FUNCTION_BLOCK PAETransport EXTENDS PAModule
VAR_INPUT
END_VAR
VAR_OUTPUT
END_VAR
VAR
	_PAPointMatIn1 : PAPoint(THIS^);
	_PAPointMatOut1 : PAPoint(THIS^);
END_VAR

METHOD FB_init : BOOL
VAR_INPUT
	bInitRetains : BOOL; // if TRUE, the retain variables are initialized (warm start / cold start)
	bInCopyCode : BOOL;  // if TRUE, the instance afterwards gets moved into the copy code (online change)
	parent : IACComponent;
END_VAR
AddPoint(_PAPointMatIn1);
AddPoint(_PAPointMatOut1);
END_METHOD

PROPERTY PUBLIC PAPointMatIn1 : IACPoint
GET
PAPointMatIn1 := _PAPointMatIn1;
END_GET
END_PROPERTY

PROPERTY PUBLIC PAPointMatOut1 : IACPoint
GET
PAPointMatOut1 := _PAPointMatOut1;
END_GET
END_PROPERTY

END_FUNCTION_BLOCK

(* stored: Version 1.1.0.1, ProductVersion 3.1.4020.12
   POU PAETransport: Id {37133530-2dd3-45c3-8f63-dc0566bbb9f0}, SpecialFunc None
   Method FB_init: Id {ea648bc8-1473-47eb-97e2-6872cc0b1ac4}
   Property PAPointMatIn1: Id {74cbe65a-12fe-472e-9ee2-f327a796bccd}
   Get Get: Id {4fa40fc4-e997-45ae-b75c-a297f4fdbbfa}
   Property PAPointMatOut1: Id {aec821b2-2d90-4d63-8726-ca7085cb5920}
   Get Get: Id {684386e5-9895-42b8-a476-1cf7fde4a347} *)
